// Mitsubishi GX Works2 project: BookEX6_15 Contact   PLC: Q13UDV

// global labels: Global
VAR_GLOBAL
  bVar0 AT M5000 : BOOL;
  abArray0 AT M5010 : ARRAY [0..49] OF BOOL;
  sStr0 AT D5000 : STRING[199];
  sStr1 AT D5100 : STRING[199];
  sStr2 AT D5200 : STRING[199];
  sStr3 AT D5300 : STRING[199];
  sStr4 AT D5400 : STRING[199];
  sStr5 AT D5500 : STRING[199];
  sStr6 AT D5600 : STRING[199];
  sStr7 AT D5700 : STRING[199];
  sStr8 AT D5800 : STRING[199];
  sStr9 AT D5900 : STRING[199];
  iVar0 AT D4500 : INT;
  iVar1 AT D4501 : INT;
  iVar2 AT D4502 : INT;
  iVar3 AT D4503 : INT;
  iVar4 AT D4504 : INT;
  iVar5 AT D4505 : INT;
  iVar6 AT D4506 : INT;
  iVar7 AT D4507 : INT;
  iVar8 AT D4508 : INT;
  iVar9 AT D4509 : INT;
  dVar0 AT D4510 : DINT;
  dVar1 AT D4512 : DINT;
  dVar2 AT D4514 : DINT;
  dVar3 AT D4516 : DINT;
  dVar4 AT D4518 : DINT;
  dVar5 AT D4520 : DINT;
  dVar6 AT D4522 : DINT;
  dVar7 AT D4524 : DINT;
  dVar8 AT D4526 : DINT;
  dVar9 AT D4528 : DINT;
  wVar0 AT D4530 : WORD;
  wVar1 AT D4531 : WORD;
  wVar2 AT D4532 : WORD;
  wVar3 AT D4533 : WORD;
  wVar4 AT D4534 : WORD;
  wVar5 AT D4535 : WORD;
  wVar6 AT D4536 : WORD;
  wVar7 AT D4537 : WORD;
  wVar8 AT D4538 : WORD;
  wVar9 AT D4539 : WORD;
  dwVar0 AT D4540 : DWORD;
  dwVar1 AT D4542 : DWORD;
  dwVar2 AT D4544 : DWORD;
  dwVar3 AT D4546 : DWORD;
  dwVar4 AT D4548 : DWORD;
  dwVar5 AT D4550 : DWORD;
  dwVar6 AT D4552 : DWORD;
  dwVar7 AT D4554 : DWORD;
  dwVar8 AT D4556 : DWORD;
  dwVar9 AT D4558 : DWORD;
  fsVar0 AT D4560 : REAL;
  fsVar1 AT D4562 : REAL;
  fsVar2 AT D4564 : REAL;
  fsVar3 AT D4566 : REAL;
  fsVar4 AT D4568 : REAL;
  fsVar5 AT D4570 : REAL;
  fsVar6 AT D4572 : REAL;
  fsVar7 AT D4574 : REAL;
  fsVar8 AT D4576 : REAL;
  fsVar9 AT D4578 : REAL;
  fdVar0 AT D4580 : LREAL;
  tTime0 AT D4620 : TIME;
  tTime1 AT D4622 : TIME;
  tTime2 AT D4624 : TIME;
  tTime3 AT D4626 : TIME;
  tTime4 AT D4628 : TIME;
  tTime5 AT D4630 : TIME;
  tTime6 AT D4632 : TIME;
  tTime7 AT D4634 : TIME;
  tTime8 AT D4636 : TIME;
  tTime9 AT D4638 : TIME;
  tTime10 AT D4640 : TIME;
  bVar1 AT M5001 : BOOL;
  bVar2 AT M5002 : BOOL;
  bVar3 AT M5003 : BOOL;
  bVar4 AT M5004 : BOOL;
  bVar5 AT M5005 : BOOL;
  bVar6 AT M5006 : BOOL;
  bVar7 AT M5007 : BOOL;
  bVar8 AT M5008 : BOOL;
  bVar9 AT M5009 : BOOL;
  abArray1 AT M5060 : ARRAY [0..49] OF BOOL;
  abArray2 AT M5110 : ARRAY [0..49] OF BOOL;
  abArray3 AT M5160 : ARRAY [0..49] OF BOOL;
  abArray4 AT M5210 : ARRAY [0..49] OF BOOL;
  abArray5 AT M5260 : ARRAY [0..49] OF BOOL;
  abArray6 AT M5310 : ARRAY [0..49] OF BOOL;
  abArray7 AT M5360 : ARRAY [0..49] OF BOOL;
  abArray8 AT M5410 : ARRAY [0..49] OF BOOL;
  abArray9 AT M5460 : ARRAY [0..49] OF BOOL;
  fdVar1 AT D4584 : LREAL;
  fdVar2 AT D4588 : LREAL;
  fdVar3 AT D4592 : LREAL;
  fdVar4 AT D4596 : LREAL;
  fdVar5 AT D4600 : LREAL;
  fdVar6 AT D4604 : LREAL;
  fdVar7 AT D4608 : LREAL;
  fdVar8 AT D4612 : LREAL;
  fdVar9 AT D4616 : LREAL;
  aSendData1 AT D100 : ARRAY [0..9] OF INT;
  aiTxData AT D4000 : ARRAY [0..99] OF INT;
  aiRxData AT D4100 : ARRAY [0..99] OF INT;
  iOpenOK AT D3900 : INT;
  iOpenERR AT D3901 : INT;
  iSendOK AT D3902 : INT;
  iSendERR AT D3903 : INT;
  iCloseOK AT D3906 : INT;
  iCloseERR AT D3907 : INT;
  iRecvOK AT D3904 : INT;
  iRecvERR AT D3905 : INT;
  aiTxData2 AT D4200 : ARRAY [0..99] OF INT;
  aiRxData2 AT D4300 : ARRAY [0..99] OF INT;
  iOpenOK2 AT D3908 : INT;
  iOpenERR2 AT D3909 : INT;
  iSendOK2 AT D3910 : INT;
  iSendERR2 AT D3911 : INT;
  iRecvOK2 AT D3912 : INT;
  iRecvERR2 AT D3913 : INT;
  iCloseOK2 AT D3914 : INT;
  iCloseERR2 AT D3915 : INT;
  iEOpenComp AT D3916 : INT;
  iEOpenReq AT D3917 : INT;
  iERecvFlag AT D3918 : INT;
  iOpenCode AT D3919 : INT;
  iSendCode AT D3920 : INT;
  iRecvCode AT D3921 : INT;
  iCloseCode AT D3922 : INT;
  iOpenCode2 AT D3923 : INT;
  iSendCode2 AT D3924 : INT;
  iRecvCode2 AT D3925 : INT;
  iCloseCode2 AT D3926 : INT;
  aRecvData1 AT D110 : ARRAY [0..9] OF INT;
  aSendData2 AT D120 : ARRAY [0..9] OF INT;
  aRecvData2 AT D130 : ARRAY [0..9] OF INT;
END_VAR
// user libraries (not included): HMI

PROGRAM ExLDP
VAR
  HMI05_1 : HMI05;
END_VAR
(* structured ladder/FBD written out as ST: instructions are called as NAME(EN, inputs, outputs); _pN, _eN, _tN stand for wires *)
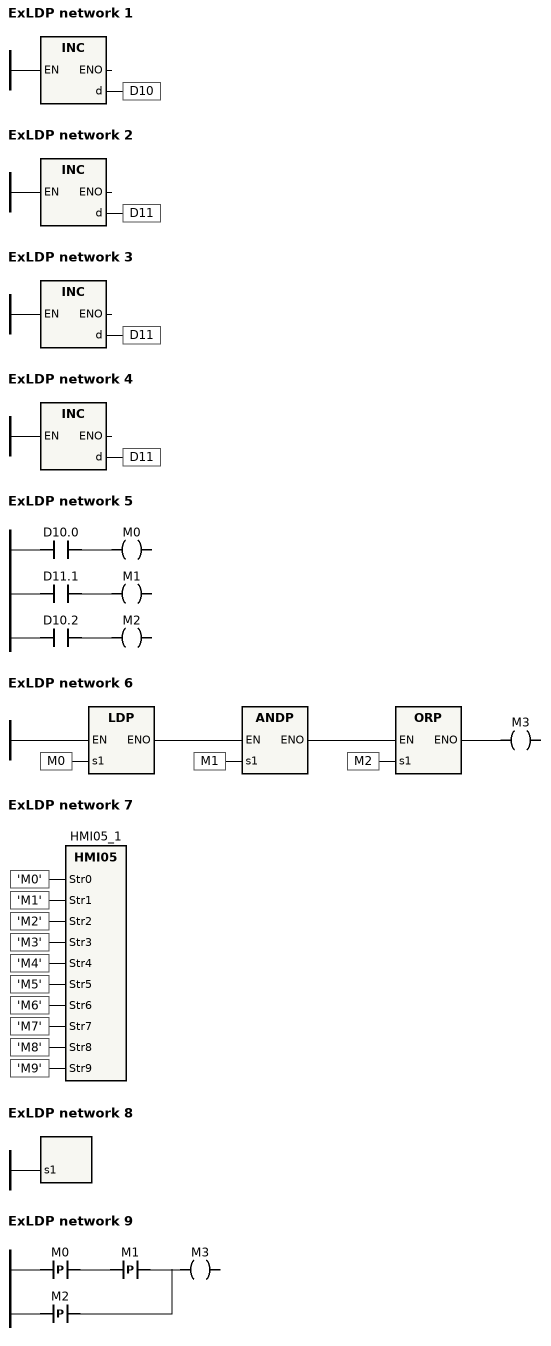
(* network 1 *)
INC(TRUE, D10);
(* network 2 *)
INC(TRUE, D11);
(* network 3 *)
INC(TRUE, D11);
(* network 4 *)
INC(TRUE, D11);
(* network 5 *)
M0 := D10.0;
M1 := D11.1;
M2 := D10.2;
(* network 6 *)
_e1 := LDP(TRUE, M0);
_e2 := ANDP(_e1, M1);
_e3 := ORP(_e2, M2);
M3 := _e3;
(* network 7 *)
HMI05_1(Str0 := 'M0', Str1 := 'M1', Str2 := 'M2', Str3 := 'M3', Str4 := 'M4', Str5 := 'M5', Str6 := 'M6', Str7 := 'M7', Str8 := 'M8', Str9 := 'M9');
(* network 8 *)
(* element kind 10  <- TRUE *)
(* network 9 *)
M3 := (LDP(TRUE, M0) AND LDP(TRUE, M1)) OR LDP(TRUE, M2);
END_PROGRAM

PROGRAM ExLDP2
VAR
  HMI05_1 : HMI05;
END_VAR
(* structured ladder/FBD written out as ST: instructions are called as NAME(EN, inputs, outputs); _pN, _eN, _tN stand for wires *)
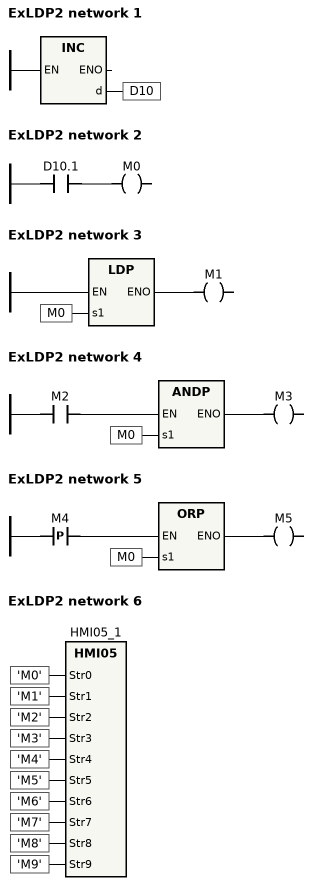
(* network 1 *)
INC(TRUE, D10);
(* network 2 *)
M0 := D10.1;
(* network 3 *)
_e1 := LDP(TRUE, M0);
M1 := _e1;
(* network 4 *)
_e1 := ANDP(M2, M0);
M3 := _e1;
(* network 5 *)
_e1 := ORP(LDP(TRUE, M4), M0);
M5 := _e1;
(* network 6 *)
HMI05_1(Str0 := 'M0', Str1 := 'M1', Str2 := 'M2', Str3 := 'M3', Str4 := 'M4', Str5 := 'M5', Str6 := 'M6', Str7 := 'M7', Str8 := 'M8', Str9 := 'M9');
END_PROGRAM

PROGRAM ExLDP3
VAR
  HMI05_1 : HMI05;
END_VAR
(* structured ladder/FBD written out as ST: instructions are called as NAME(EN, inputs, outputs); _pN, _eN, _tN stand for wires *)
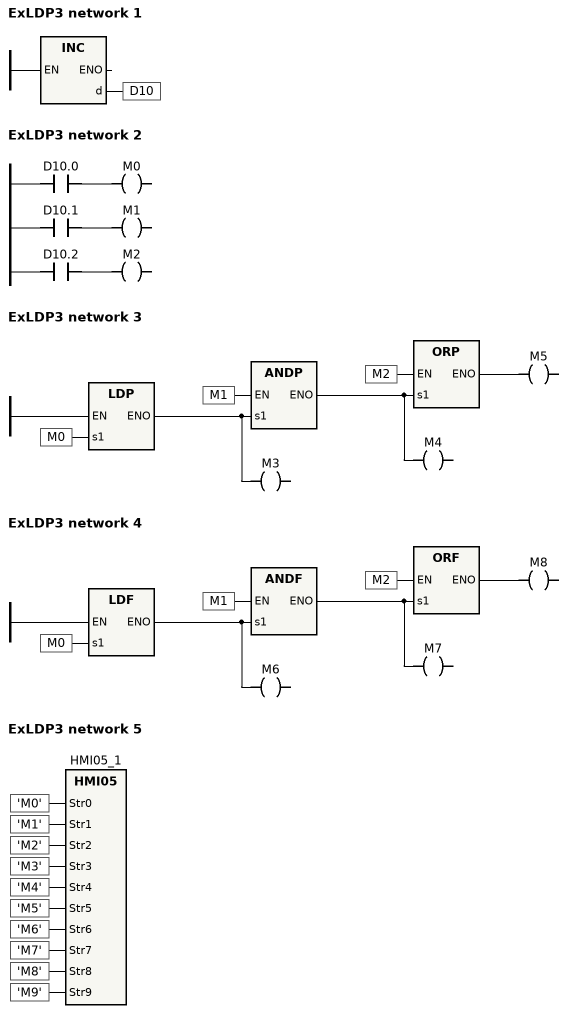
(* network 1 *)
INC(TRUE, D10);
(* network 2 *)
M0 := D10.0;
M1 := D10.1;
M2 := D10.2;
(* network 3 *)
_e1 := LDP(TRUE, M0);
_e2 := ANDP(M1, _e1);
_e3 := ORP(M2, _e2);
M5 := _e3;
M4 := _e2;
M3 := _e1;
(* network 4 *)
_e1 := LDF(TRUE, M0);
_e2 := ANDF(M1, _e1);
_e3 := ORF(M2, _e2);
M8 := _e3;
M7 := _e2;
M6 := _e1;
(* network 5 *)
HMI05_1(Str0 := 'M0', Str1 := 'M1', Str2 := 'M2', Str3 := 'M3', Str4 := 'M4', Str5 := 'M5', Str6 := 'M6', Str7 := 'M7', Str8 := 'M8', Str9 := 'M9');
END_PROGRAM

PROGRAM ExLDPI
VAR
  HMI05_1 : HMI05;
END_VAR
(* structured ladder/FBD written out as ST: instructions are called as NAME(EN, inputs, outputs); _pN, _eN, _tN stand for wires *)
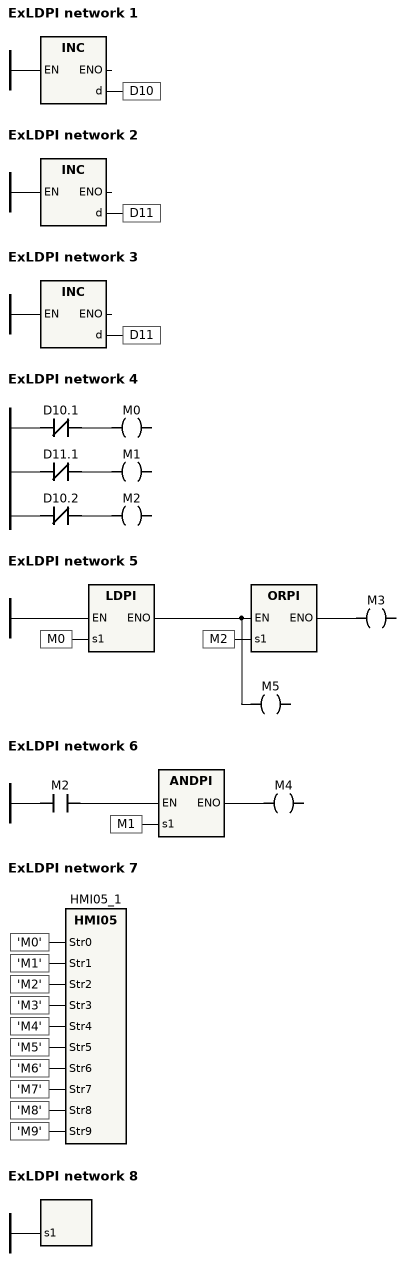
(* network 1 *)
INC(TRUE, D10);
(* network 2 *)
INC(TRUE, D11);
(* network 3 *)
INC(TRUE, D11);
(* network 4 *)
M0 := NOT D10.1;
M1 := NOT D11.1;
M2 := NOT D10.2;
(* network 5 *)
_e1 := LDPI(TRUE, M0);
M5 := _e1;
_e2 := ORPI(_e1, M2);
M3 := _e2;
(* network 6 *)
_e1 := ANDPI(M2, M1);
M4 := _e1;
(* network 7 *)
HMI05_1(Str0 := 'M0', Str1 := 'M1', Str2 := 'M2', Str3 := 'M3', Str4 := 'M4', Str5 := 'M5', Str6 := 'M6', Str7 := 'M7', Str8 := 'M8', Str9 := 'M9');
(* network 8 *)
(* element kind 10  <- TRUE *)
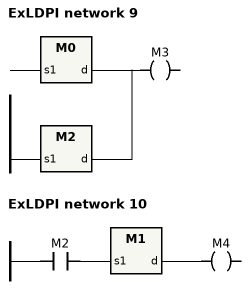
(* network 9 *)
(* element kind 19 M0 <- TRUE *)
(* element kind 19 M2 <- TRUE *)
M3 := _feedback OR _feedback;
(* network 10 *)
(* element kind 19 M1 <- M2 *)
M4 := _feedback;
END_PROGRAM

PROGRAM ExLDPI2
VAR
  HMI05_1 : HMI05;
END_VAR
(* structured ladder/FBD written out as ST: instructions are called as NAME(EN, inputs, outputs); _pN, _eN, _tN stand for wires *)
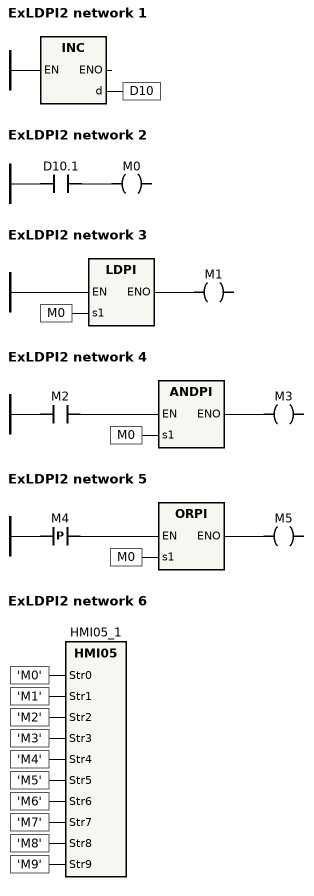
(* network 1 *)
INC(TRUE, D10);
(* network 2 *)
M0 := D10.1;
(* network 3 *)
_e1 := LDPI(TRUE, M0);
M1 := _e1;
(* network 4 *)
_e1 := ANDPI(M2, M0);
M3 := _e1;
(* network 5 *)
_e1 := ORPI(LDP(TRUE, M4), M0);
M5 := _e1;
(* network 6 *)
HMI05_1(Str0 := 'M0', Str1 := 'M1', Str2 := 'M2', Str3 := 'M3', Str4 := 'M4', Str5 := 'M5', Str6 := 'M6', Str7 := 'M7', Str8 := 'M8', Str9 := 'M9');
END_PROGRAM

PROGRAM ExLDPI3
VAR
  HMI05_1 : HMI05;
END_VAR
(* structured ladder/FBD written out as ST: instructions are called as NAME(EN, inputs, outputs); _pN, _eN, _tN stand for wires *)
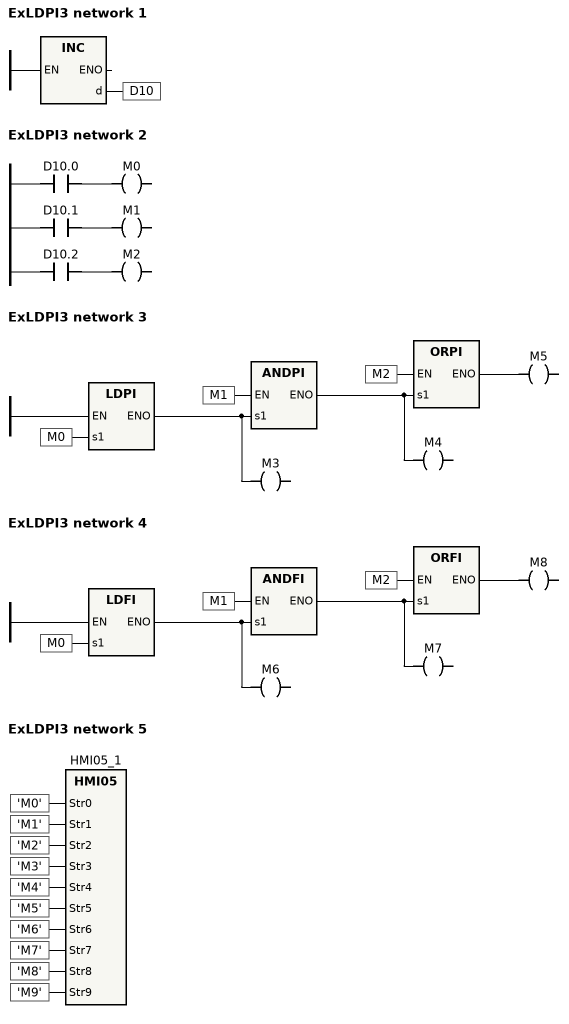
(* network 1 *)
INC(TRUE, D10);
(* network 2 *)
M0 := D10.0;
M1 := D10.1;
M2 := D10.2;
(* network 3 *)
_e1 := LDPI(TRUE, M0);
_e2 := ANDPI(M1, _e1);
_e3 := ORPI(M2, _e2);
M5 := _e3;
M4 := _e2;
M3 := _e1;
(* network 4 *)
_e1 := LDFI(TRUE, M0);
_e2 := ANDFI(M1, _e1);
_e3 := ORFI(M2, _e2);
M8 := _e3;
M7 := _e2;
M6 := _e1;
(* network 5 *)
HMI05_1(Str0 := 'M0', Str1 := 'M1', Str2 := 'M2', Str3 := 'M3', Str4 := 'M4', Str5 := 'M5', Str6 := 'M6', Str7 := 'M7', Str8 := 'M8', Str9 := 'M9');
END_PROGRAM

PROGRAM Sample
(* structured ladder/FBD written out as ST: instructions are called as NAME(EN, inputs, outputs); _pN, _eN, _tN stand for wires *)
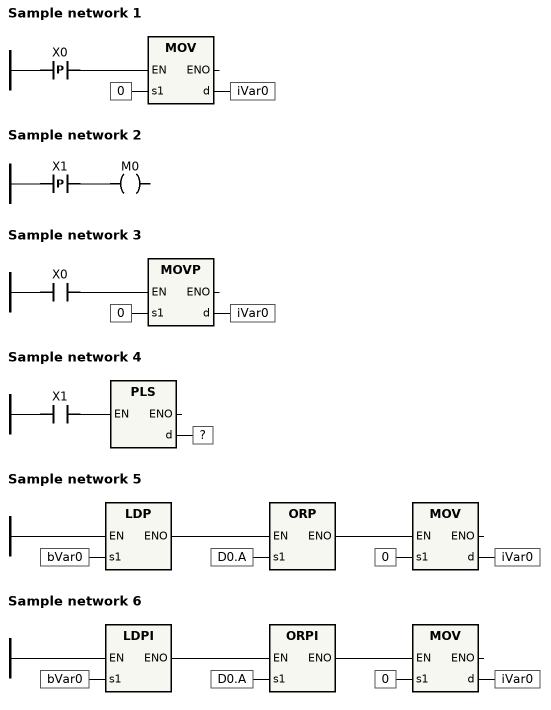
(* network 1 *)
MOV(LDP(TRUE, X0), 0, iVar0);
(* network 2 *)
M0 := LDP(TRUE, X1);
(* network 3 *)
MOVP(X0, 0, iVar0);
(* network 4 *)
PLS(X1, ?);
(* network 5 *)
_e1 := LDP(TRUE, bVar0);
_e2 := ORP(_e1, D0.A);
MOV(_e2, 0, iVar0);
(* network 6 *)
_e1 := LDPI(TRUE, bVar0);
_e2 := ORPI(_e1, D0.A);
MOV(_e2, 0, iVar0);
END_PROGRAM

PROGRAM ExLDP4
(* structured ladder/FBD written out as ST: instructions are called as NAME(EN, inputs, outputs); _pN, _eN, _tN stand for wires *)
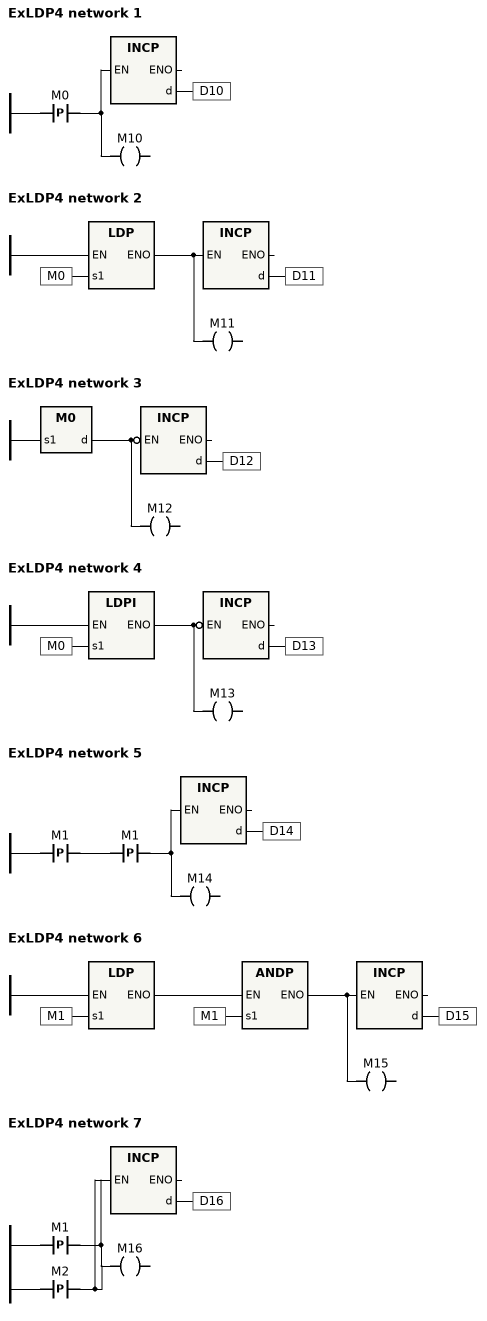
(* network 1 *)
_p1 := LDP(TRUE, M0);
INCP(_p1, D10);
M10 := _p1;
(* network 2 *)
_e1 := LDP(TRUE, M0);
INCP(_e1, D11);
M11 := _e1;
(* network 3 *)
(* element kind 19 M0 <- TRUE *)
INCP(NOT _feedback, D12);
M12 := _feedback;
(* network 4 *)
_e1 := LDPI(TRUE, M0);
INCP(NOT _e1, D13);
M13 := _e1;
(* network 5 *)
_p1 := LDP(TRUE, M1) AND LDP(TRUE, M1);
INCP(_p1, D14);
M14 := _p1;
(* network 6 *)
_e1 := LDP(TRUE, M1);
_e2 := ANDP(_e1, M1);
INCP(_e2, D15);
M15 := _e2;
(* network 7 *)
_p1 := LDP(TRUE, M1) OR LDP(TRUE, M2);
INCP(_p1, D16);
M16 := _p1;
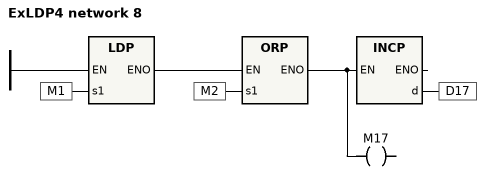
(* network 8 *)
_e1 := LDP(TRUE, M1);
_e2 := ORP(_e1, M2);
INCP(_e2, D17);
M17 := _e2;
END_PROGRAM
